// TIA Portal V15.1 export
// export: Created 2024-06-21T08:41:13.9396276Z, ExportSetting WithDefaults, DisplayName Totally Integrated Automation Portal, DisplayVersion V15.1 Update 5, DisplayName TIA Portal Openness, DisplayVersion V15.1 Update 5, DisplayName SINAMICS Startdrive Advanced, DisplayVersion V15.1, DisplayName G130, G150, S120, S150, SINAMICS MV, S210, DisplayVersion V15.1, DisplayName G110M, G120, G120C, G120D, G120P, DisplayVersion V15.1, DisplayName STEP 7 Professional, DisplayVersion V15.1 Update 5, DisplayName STEP 7 Safety, DisplayVersion V15.1, DisplayName WinCC Professional, DisplayVersion V15.1 Update 5, DisplayName SIMATIC Visualization Architect, DisplayVersion V15.1
FUNCTION_BLOCK "LGBBuhlLock"   // FB6630, FBD
TITLE = LGBBuhlLock
{ S7_Optimized_Access := 'TRUE' }
AUTHOR : VCC
FAMILY : Tooling
VERSION : 0.1
// ==================================================
// This module handles a Move Unit with 2 Positions and Contactor
// ==================================================
// stored: AutoNumber false, IsIECCheckEnabled false, IsRetainMemResEnabled false, MemoryReserve 100, SetENOAutomatically False, UDAEnableTagReadback false
   VAR_INPUT
      I_PosSetDet1 { ExternalAccessible := 'False'; ExternalVisible := 'False'; ExternalWritable := 'False'} : Bool;   // Position Set Detection1 (Unlocked)
      I_PosSetDet2 { ExternalAccessible := 'False'; ExternalVisible := 'False'; ExternalWritable := 'False'} : Bool;   // Position Set Detection2 (Unlocked)
      I_PosResDet1 { ExternalAccessible := 'False'; ExternalVisible := 'False'; ExternalWritable := 'False'} : Bool;   // Position Reset Detection1 (Locked)
      I_PosResDet2 { ExternalAccessible := 'False'; ExternalVisible := 'False'; ExternalWritable := 'False'} : Bool;   // Position Reset Detection2 (Locked)
      I_Ready { ExternalAccessible := 'False'; ExternalVisible := 'False'; ExternalWritable := 'False'} : Bool;   // Device Ready
      I_SetBegin { ExternalAccessible := 'False'; ExternalVisible := 'False'; ExternalWritable := 'False'} : Bool;   // Function Set begin selection
      I_ResBegin { ExternalAccessible := 'False'; ExternalVisible := 'False'; ExternalWritable := 'False'} : Bool;   // Function Reset begin selection
      I_PBSet { ExternalAccessible := 'False'; ExternalVisible := 'False'; ExternalWritable := 'False'} : Bool;   // Push button for Set direction (used in manual with button OP panels )
      I_PBReset { ExternalAccessible := 'False'; ExternalVisible := 'False'; ExternalWritable := 'False'} : Bool;   // Push button for Reset direction (used in manual with Pushbutton OP panels)
      I_SetIntlkOK { ExternalAccessible := 'False'; ExternalVisible := 'False'; ExternalWritable := 'False'} : Bool;   // Set Interlock
      I_ResIntlkOK { ExternalAccessible := 'False'; ExternalVisible := 'False'; ExternalWritable := 'False'} : Bool;   // Reset Interlock
      I_SafetyOk { ExternalAccessible := 'False'; ExternalVisible := 'False'; ExternalWritable := 'False'} : Bool;   // Safety Ok
      I_MotorProtection { ExternalAccessible := 'False'; ExternalVisible := 'False'; ExternalWritable := 'False'} : Bool;   // Motor protection
      I_SafetySwitch { ExternalAccessible := 'False'; ExternalVisible := 'False'; ExternalWritable := 'False'} : Bool;   // Safety Switch
      I_ModeScreenChanged { ExternalAccessible := 'False'; ExternalVisible := 'False'; ExternalWritable := 'False'} : Bool;   // Screen Changed
   END_VAR
   VAR_OUTPUT
      O_CmdSet { ExternalAccessible := 'False'; ExternalVisible := 'False'; ExternalWritable := 'False'} : Bool;   // Command to Activate Set movement
      O_CmdRes { ExternalAccessible := 'False'; ExternalVisible := 'False'; ExternalWritable := 'False'} : Bool;   // Command to Activate Reset movement
      O_SumPosSet { ExternalAccessible := 'False'; ExternalVisible := 'False'; ExternalWritable := 'False'} : Bool;   // Summary In Position Set
      O_SumPosRes { ExternalAccessible := 'False'; ExternalVisible := 'False'; ExternalWritable := 'False'} : Bool;   // Summary In Position Reset
      O_FuncRunning { ExternalAccessible := 'False'; ExternalVisible := 'False'; ExternalWritable := 'False'} : Bool;   // Signal that the function is busy
      O_SetFinished { ExternalAccessible := 'False'; ExternalVisible := 'False'; ExternalWritable := 'False'} : Bool;   // Function Set finished
      O_ResFinished { ExternalAccessible := 'False'; ExternalVisible := 'False'; ExternalWritable := 'False'} : Bool;   // Function Reset finished
      O_AlarmABCondition { ExternalAccessible := 'False'; ExternalVisible := 'False'; ExternalWritable := 'False'} : Bool;   // Alarm AB Condition
      O_AlarmA { ExternalAccessible := 'False'; ExternalVisible := 'False'; ExternalWritable := 'False'} : Bool;   // Alarm A
      O_AlarmB { ExternalAccessible := 'False'; ExternalVisible := 'False'; ExternalWritable := 'False'} : Bool;   // Alarm B
      O_AlarmC { ExternalAccessible := 'False'; ExternalVisible := 'False'; ExternalWritable := 'False'} : Bool;   // Alarm C
      O_AlarmD { ExternalAccessible := 'False'; ExternalVisible := 'False'; ExternalWritable := 'False'} : Bool;   // Alarm D
      H_AlarmDWord { ExternalAccessible := 'False'; ExternalVisible := 'False'; ExternalWritable := 'False'} : DWord;   // HMI Alarm Word
   END_VAR
   VAR_IN_OUT
      IO_ModeSelector : Struct   // Mode Selector
         AutoSel : Bool;
         AllAutoSel : Bool;
         StepSel : Bool;
         HomeRunSel : Bool;
         ManualSel : Bool;
         ForcedManActSel : Bool;
         PBSetSel : Bool;
         PBResetSel : Bool;
         StartPBSel : Bool;
         AlarmResetPBSel : Bool;
         ResetTMSel : Bool;
         ResetSeqSel : Bool;
         CycleFinishedSel : Bool;
         HomeRunRedoSel : Bool;
         HomeRunWorkDoneSel : Bool;
         ResetSafetyInputSel : Bool;
      END_STRUCT;
      IO_Alarm : "Alarm";   // Alarm
      C_MovConfig : "MovConfig";   // Config
      H_HMI : "H_HMI";   // Animation
      H_GBBuhlLock : "H_GBBuhlLock";   // Animation
   END_VAR
   VAR
      Modes { ExternalAccessible := 'False'; ExternalVisible := 'False'; ExternalWritable := 'False'} : "Modes";   // Modes
      H_FncSelInHMI { ExternalAccessible := 'False'; ExternalVisible := 'False'; ExternalWritable := 'False'} : Bool;
      AA_MotorProtection { ExternalAccessible := 'False'; ExternalVisible := 'False'; ExternalWritable := 'False'} : Bool;   // Motorprotection Not Ok / Motorprotection Tripped
      AA_SafetySwitch { ExternalAccessible := 'False'; ExternalVisible := 'False'; ExternalWritable := 'False'} : Bool;   // Safety Switch Not Ok
      AB_KeepPosSetAlm { ExternalAccessible := 'False'; ExternalVisible := 'False'; ExternalWritable := 'False'} : Bool;   // Lost Set Position / Alarm Keep Position Set
      AB_KeepPosResAlm { ExternalAccessible := 'False'; ExternalVisible := 'False'; ExternalWritable := 'False'} : Bool;   // Lost Reset Position / Alarm Keep Position Reset
      AB_OvtSetAlm { ExternalAccessible := 'False'; ExternalVisible := 'False'; ExternalWritable := 'False'} : Bool;   // TimeOut Set Direction / Timeout Set
      AB_OvtResAlm { ExternalAccessible := 'False'; ExternalVisible := 'False'; ExternalWritable := 'False'} : Bool;   // TimeOut Reset Direction / Timeout Reset
      AB_TwoDetAlm { ExternalAccessible := 'False'; ExternalVisible := 'False'; ExternalWritable := 'False'} : Bool;   // Detection Set & Reset Activated Simultaneously / Set Reset Activated Simultaneously
      AC_KeepPosSetAlm { ExternalAccessible := 'False'; ExternalVisible := 'False'; ExternalWritable := 'False'} : Bool;   // Lost Set Position / Alarm Keep Position Set
      AC_KeepPosResAlm { ExternalAccessible := 'False'; ExternalVisible := 'False'; ExternalWritable := 'False'} : Bool;   // Lost Reset Position / Alarm Keep Position Reset
      AC_OvtSetAlm { ExternalAccessible := 'False'; ExternalVisible := 'False'; ExternalWritable := 'False'} : Bool;   // TimeOut Set Direction / Timeout Set
      AC_OvtResAlm { ExternalAccessible := 'False'; ExternalVisible := 'False'; ExternalWritable := 'False'} : Bool;   // TimeOut Reset Direction / Timeout Reset
      AC_TwoDetAlm { ExternalAccessible := 'False'; ExternalVisible := 'False'; ExternalWritable := 'False'} : Bool;   // Detection Set & Reset Activated Simultaneously / Set Reset Activated Simultaneously
      AD_OvtSetWarn { ExternalAccessible := 'False'; ExternalVisible := 'False'; ExternalWritable := 'False'} : Bool;   // TimeOut Set Direction / Timeout Set
      AD_OvtResWarn { ExternalAccessible := 'False'; ExternalVisible := 'False'; ExternalWritable := 'False'} : Bool;   // TimeOut Reset Direction / Timeout Reset
      AD_IntlkSetAlm { ExternalAccessible := 'False'; ExternalVisible := 'False'; ExternalWritable := 'False'} : Bool;   // Interlock Set
      AD_IntlkResAlm { ExternalAccessible := 'False'; ExternalVisible := 'False'; ExternalWritable := 'False'} : Bool;   // Interlock Reset
      AC_NotReadyAlm { ExternalAccessible := 'False'; ExternalVisible := 'False'; ExternalWritable := 'False'} : Bool;   // Not Ready To Run
      AC_ConfigCalibrationAlm { ExternalAccessible := 'False'; ExternalVisible := 'False'; ExternalWritable := 'False'} : Bool;   // The Config values for Warming/Alarm time must be ALL zero or ALL different from zero
      AD_CalibrationWarn { ExternalAccessible := 'False'; ExternalVisible := 'False'; ExternalWritable := 'False'} : Bool;   // No High speed selected so Calibration is not possible
      CmdSet { ExternalAccessible := 'False'; ExternalVisible := 'False'; ExternalWritable := 'False'} : Bool;   // Command set
      CmdRes { ExternalAccessible := 'False'; ExternalVisible := 'False'; ExternalWritable := 'False'} : Bool;   // DCommand Reset
      SetPos { ExternalAccessible := 'False'; ExternalVisible := 'False'; ExternalWritable := 'False'} : Bool;   // Set Position
      ResPos { ExternalAccessible := 'False'; ExternalVisible := 'False'; ExternalWritable := 'False'} : Bool;   // Reset Position
      AlarmA { ExternalAccessible := 'False'; ExternalVisible := 'False'; ExternalWritable := 'False'} : Bool;   // Summation Alarm A
      AlarmB { ExternalAccessible := 'False'; ExternalVisible := 'False'; ExternalWritable := 'False'} : Bool;   // Summation Alarm B
      AlarmC { ExternalAccessible := 'False'; ExternalVisible := 'False'; ExternalWritable := 'False'} : Bool;   // Summation Alarm C
      AlarmD { ExternalAccessible := 'False'; ExternalVisible := 'False'; ExternalWritable := 'False'} : Bool;   // Summation Alarm D
      FuncRunning { ExternalAccessible := 'False'; ExternalVisible := 'False'; ExternalWritable := 'False'} : Bool;   // Function running
      MovFuncAlmCond { ExternalAccessible := 'False'; ExternalVisible := 'False'; ExternalWritable := 'False'} : Bool;   // Move function Alarm Condition
      StopPosAlmCond { ExternalAccessible := 'False'; ExternalVisible := 'False'; ExternalWritable := 'False'} : Bool;   // Stop posistion Alarm Condition
      KeepPosSetAlm { ExternalAccessible := 'False'; ExternalVisible := 'False'; ExternalWritable := 'False'} : Bool;   // Keep Position Set Alarm
      KeepPosResAlm { ExternalAccessible := 'False'; ExternalVisible := 'False'; ExternalWritable := 'False'} : Bool;   // Keep Position Reset Alarm
      OvtSetAlm { ExternalAccessible := 'False'; ExternalVisible := 'False'; ExternalWritable := 'False'} : Bool;   // Overtime set Alarm
      OvtResAlm { ExternalAccessible := 'False'; ExternalVisible := 'False'; ExternalWritable := 'False'} : Bool;   // Overtime Reset Alarm
      TwoDetAlm { ExternalAccessible := 'False'; ExternalVisible := 'False'; ExternalWritable := 'False'} : Bool;   // Two detection Alarm
      OutOfUse { ExternalAccessible := 'False'; ExternalVisible := 'False'; ExternalWritable := 'False'} : Bool;   // Out of use
      AlarmABCondition { ExternalAccessible := 'False'; ExternalVisible := 'False'; ExternalWritable := 'False'} : Bool;   // Alarm AB Condition
      ContactorSet { ExternalAccessible := 'False'; ExternalVisible := 'False'; ExternalWritable := 'False'} : Bool;   // Contactor Set
      ContactorRes { ExternalAccessible := 'False'; ExternalVisible := 'False'; ExternalWritable := 'False'} : Bool;   // Contactor Reset
      MotorLoopAlmCond { ExternalAccessible := 'False'; ExternalVisible := 'False'; ExternalWritable := 'False'} : Bool;   // Motor loop Alarm condition
      MotorLoopActive { ExternalAccessible := 'False'; ExternalVisible := 'False'; ExternalWritable := 'False'} : Bool;   // Motor Loop Active
      ManReqSet { ExternalAccessible := 'False'; ExternalVisible := 'False'; ExternalWritable := 'False'} : Bool;   // In Manual AND Request Maintenance door
      ManReqReset { ExternalAccessible := 'False'; ExternalVisible := 'False'; ExternalWritable := 'False'} : Bool;   // In Manual AND No Request Maintenance door
      MovFunc2Pos { ExternalAccessible := 'False'; ExternalVisible := 'False'; ExternalWritable := 'False'} : "LMovFnc2Pos";   // FB
      StopPos { ExternalAccessible := 'False'; ExternalVisible := 'False'; ExternalWritable := 'False'} : "L2StopPos";   // FB
      _Motor { ExternalAccessible := 'False'; ExternalVisible := 'False'; ExternalWritable := 'False'} : "LGBMotor2W1S-C";   // FB
      PosSetDelayTimer { ExternalAccessible := 'False'; ExternalVisible := 'False'; ExternalWritable := 'False'} : "LTimer";   // FB
      PosResDelayTimer { ExternalAccessible := 'False'; ExternalVisible := 'False'; ExternalWritable := 'False'} : "LTimer";   // FB
      TP_ManReqSet { ExternalAccessible := 'False'; ExternalVisible := 'False'; ExternalWritable := 'False'} : TP_TIME;   // Timer
      TP_ManReqReset { ExternalAccessible := 'False'; ExternalVisible := 'False'; ExternalWritable := 'False'} : TP_TIME;   // Timer
   END_VAR
   VAR_TEMP
      H_HMITemp : "H_HMI";   // Temp
   END_VAR
   VAR_TEMP   // added for the SCL form of the ladder/FBD networks
      _w1 : Bool;
   END_VAR
BEGIN

REGION Network 1: **** 1 - Inputs **** HMI Commands
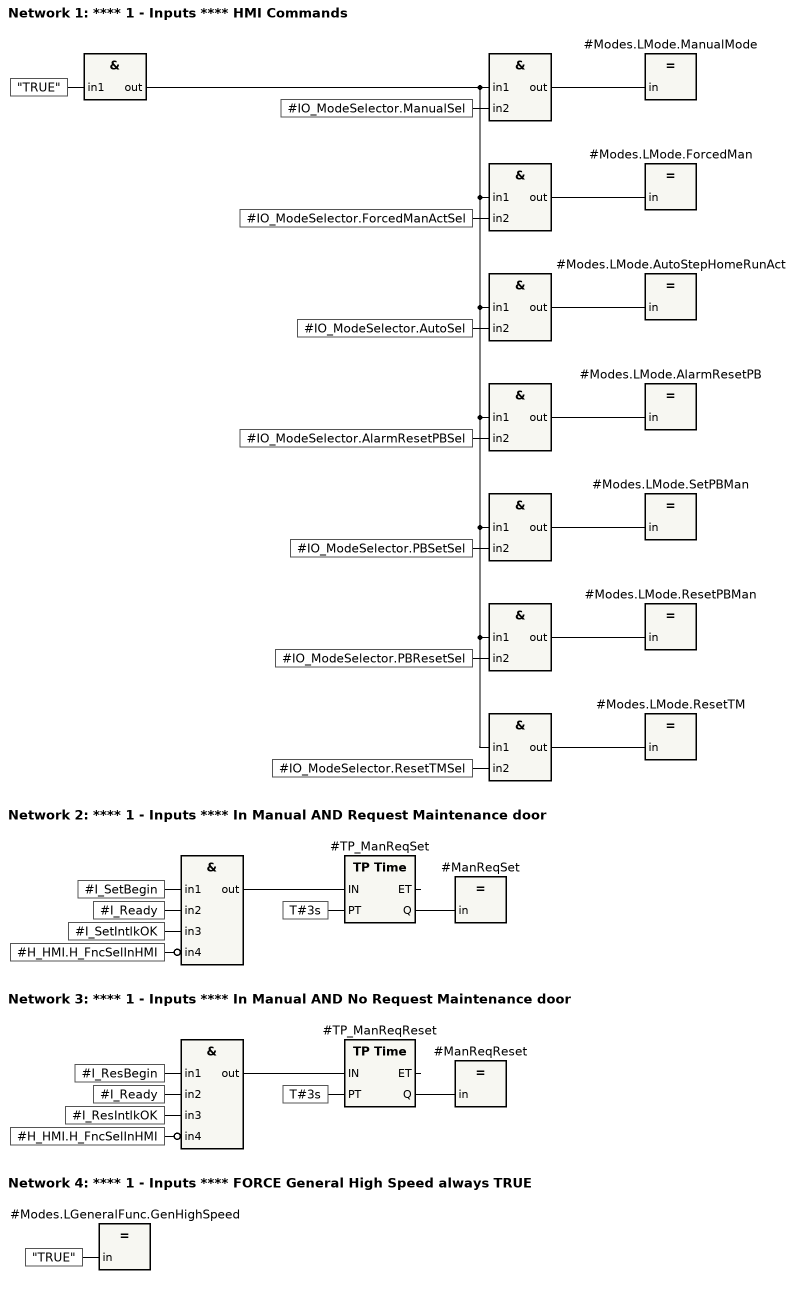
   #Modes.LMode.ManualMode := "TRUE" AND #IO_ModeSelector.ManualSel;
   #Modes.LMode.ForcedMan := "TRUE" AND #IO_ModeSelector.ForcedManActSel;
   #Modes.LMode.AutoStepHomeRunAct := "TRUE" AND #IO_ModeSelector.AutoSel;
   #Modes.LMode.AlarmResetPB := "TRUE" AND #IO_ModeSelector.AlarmResetPBSel;
   #Modes.LMode.SetPBMan := "TRUE" AND #IO_ModeSelector.PBSetSel;
   #Modes.LMode.ResetPBMan := "TRUE" AND #IO_ModeSelector.PBResetSel;
   #Modes.LMode.ResetTM := "TRUE" AND #IO_ModeSelector.ResetTMSel;
END_REGION

REGION Network 2: **** 1 - Inputs **** In Manual AND Request Maintenance door
   #TP_ManReqSet(IN := #I_SetBegin AND #I_Ready AND #I_SetIntlkOK AND NOT #H_HMI.H_FncSelInHMI, PT := T#3s);   // TP
   #ManReqSet := #TP_ManReqSet.Q;
END_REGION

REGION Network 3: **** 1 - Inputs **** In Manual AND No Request Maintenance door
   #TP_ManReqReset(IN := #I_ResBegin AND #I_Ready AND #I_ResIntlkOK AND NOT #H_HMI.H_FncSelInHMI, PT := T#3s);   // TP
   #ManReqReset := #TP_ManReqReset.Q;
END_REGION

REGION Network 4: **** 1 - Inputs **** FORCE General High Speed always TRUE
   #Modes.LGeneralFunc.GenHighSpeed := "TRUE";
END_REGION

REGION Network 5: **** 2.2 - Alarms - Alarm Generation **** Two Detection B Alarm
   // Two Detection B Alarm
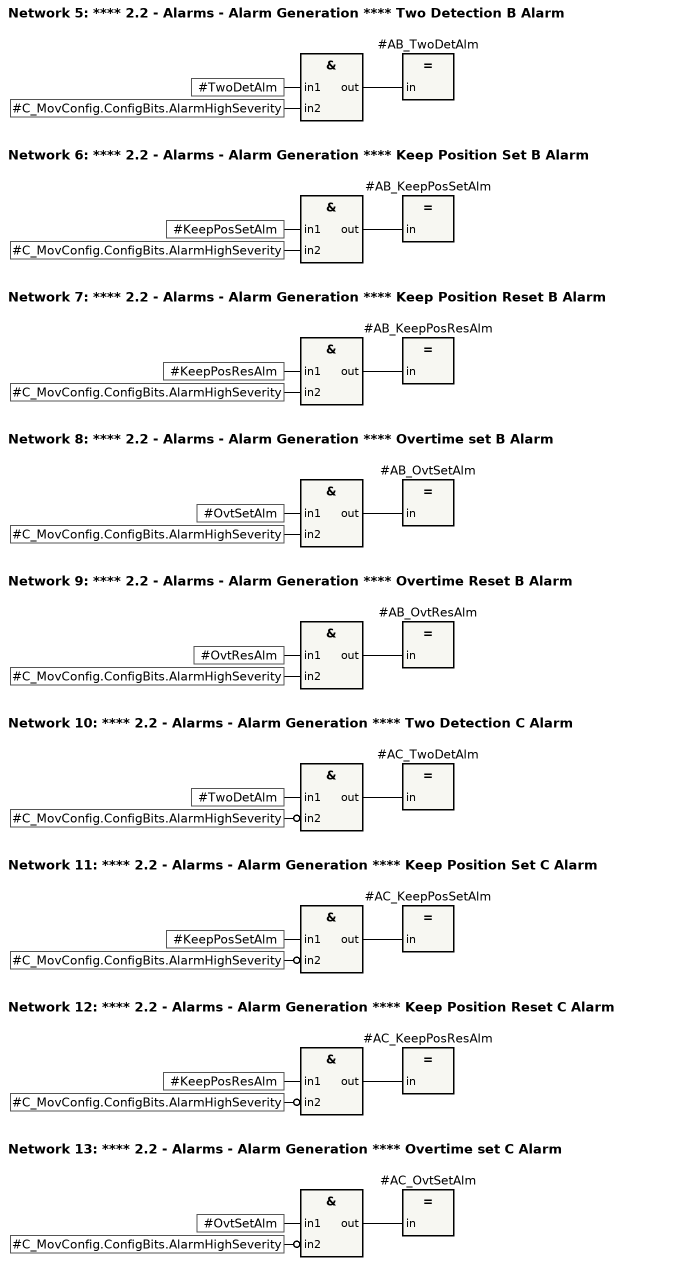
   #AB_TwoDetAlm := #TwoDetAlm AND #C_MovConfig.ConfigBits.AlarmHighSeverity;
END_REGION

REGION Network 6: **** 2.2 - Alarms - Alarm Generation **** Keep Position Set B Alarm
   // Keep Position Set B Alarm
   #AB_KeepPosSetAlm := #KeepPosSetAlm AND #C_MovConfig.ConfigBits.AlarmHighSeverity;
END_REGION

REGION Network 7: **** 2.2 - Alarms - Alarm Generation **** Keep Position Reset B Alarm
   // Keep Position Reset B Alarm
   #AB_KeepPosResAlm := #KeepPosResAlm AND #C_MovConfig.ConfigBits.AlarmHighSeverity;
END_REGION

REGION Network 8: **** 2.2 - Alarms - Alarm Generation **** Overtime set B Alarm
   // Overtime set B Alarm
   #AB_OvtSetAlm := #OvtSetAlm AND #C_MovConfig.ConfigBits.AlarmHighSeverity;
END_REGION

REGION Network 9: **** 2.2 - Alarms - Alarm Generation **** Overtime Reset B Alarm
   // Overtime Reset B Alarm
   #AB_OvtResAlm := #OvtResAlm AND #C_MovConfig.ConfigBits.AlarmHighSeverity;
END_REGION

REGION Network 10: **** 2.2 - Alarms - Alarm Generation **** Two Detection C Alarm
   // Two Detection C Alarm
   #AC_TwoDetAlm := #TwoDetAlm AND NOT #C_MovConfig.ConfigBits.AlarmHighSeverity;
END_REGION

REGION Network 11: **** 2.2 - Alarms - Alarm Generation **** Keep Position Set C Alarm
   // Keep Position Set C Alarm
   #AC_KeepPosSetAlm := #KeepPosSetAlm AND NOT #C_MovConfig.ConfigBits.AlarmHighSeverity;
END_REGION

REGION Network 12: **** 2.2 - Alarms - Alarm Generation **** Keep Position Reset C Alarm
   // Keep Position Reset C Alarm
   #AC_KeepPosResAlm := #KeepPosResAlm AND NOT #C_MovConfig.ConfigBits.AlarmHighSeverity;
END_REGION

REGION Network 13: **** 2.2 - Alarms - Alarm Generation **** Overtime set C Alarm
   // Overtime set C Alarm
   #AC_OvtSetAlm := #OvtSetAlm AND NOT #C_MovConfig.ConfigBits.AlarmHighSeverity;
END_REGION

REGION Network 14: **** 2.2 - Alarms - Alarm Generation **** Overtime Reset C Alarm
   // Overtime Reset C Alarm
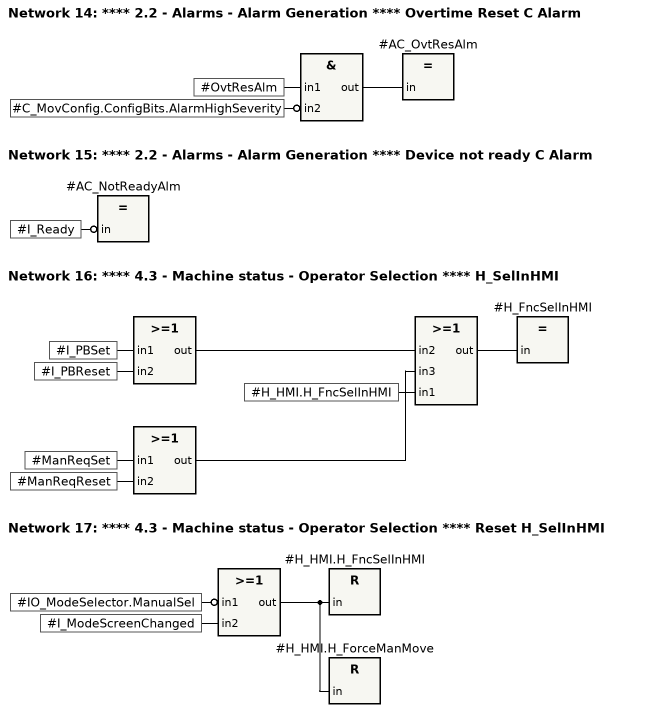
   #AC_OvtResAlm := #OvtResAlm AND NOT #C_MovConfig.ConfigBits.AlarmHighSeverity;
END_REGION

REGION Network 15: **** 2.2 - Alarms - Alarm Generation **** Device not ready C Alarm
   // Device not ready C Alarm
   #AC_NotReadyAlm := NOT #I_Ready;
END_REGION

REGION Network 16: **** 4.3 - Machine status - Operator Selection **** H_SelInHMI
   #H_FncSelInHMI := #I_PBSet OR #I_PBReset OR #ManReqSet OR #ManReqReset OR #H_HMI.H_FncSelInHMI;
END_REGION

REGION Network 17: **** 4.3 - Machine status - Operator Selection **** Reset H_SelInHMI
   // Reset H_SelInHMI
   IF NOT #IO_ModeSelector.ManualSel OR #I_ModeScreenChanged THEN
       #H_HMI.H_FncSelInHMI := FALSE;
       #H_HMI.H_ForceManMove := FALSE;
   END_IF;
END_REGION

REGION Network 18: **** 4.6 - Machine Status - Indication **** Icon Animation
   // Icon Animation
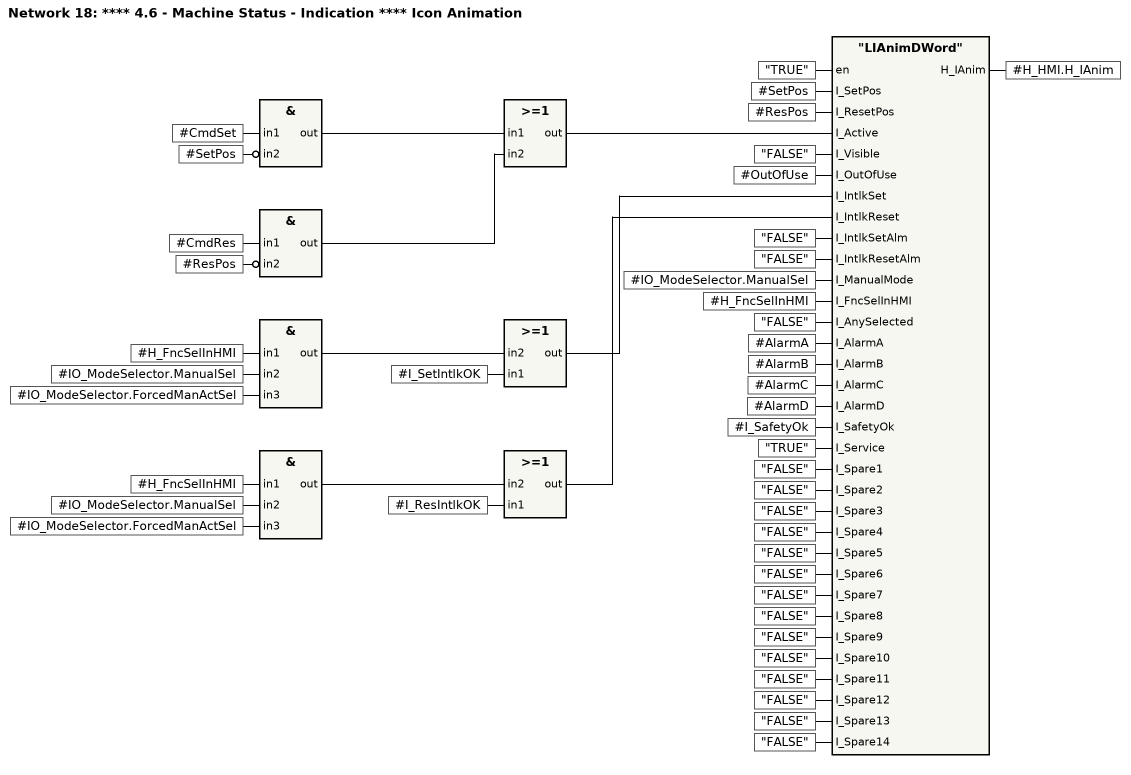
   IF "TRUE" THEN
       "LIAnimDWord"(I_SetPos := #SetPos,
                     I_ResetPos := #ResPos,
                     I_Active := (#CmdSet AND NOT #SetPos) OR (#CmdRes AND NOT #ResPos),
                     I_Visible := "FALSE",
                     I_OutOfUse := #OutOfUse,
                     I_IntlkSet := (#H_FncSelInHMI AND #IO_ModeSelector.ManualSel AND #IO_ModeSelector.ForcedManActSel) OR #I_SetIntlkOK,
                     I_IntlkReset := (#H_FncSelInHMI AND #IO_ModeSelector.ManualSel AND #IO_ModeSelector.ForcedManActSel) OR #I_ResIntlkOK,
                     I_IntlkSetAlm := "FALSE",
                     I_IntlkResetAlm := "FALSE",
                     I_ManualMode := #IO_ModeSelector.ManualSel,
                     I_FncSelInHMI := #H_FncSelInHMI,
                     I_AnySelected := "FALSE",
                     I_AlarmA := #AlarmA,
                     I_AlarmB := #AlarmB,
                     I_AlarmC := #AlarmC,
                     I_AlarmD := #AlarmD,
                     I_SafetyOk := #I_SafetyOk,
                     I_Service := "TRUE",
                     I_Spare1 := "FALSE",
                     I_Spare2 := "FALSE",
                     I_Spare3 := "FALSE",
                     I_Spare4 := "FALSE",
                     I_Spare5 := "FALSE",
                     I_Spare6 := "FALSE",
                     I_Spare7 := "FALSE",
                     I_Spare8 := "FALSE",
                     I_Spare9 := "FALSE",
                     I_Spare10 := "FALSE",
                     I_Spare11 := "FALSE",
                     I_Spare12 := "FALSE",
                     I_Spare13 := "FALSE",
                     I_Spare14 := "FALSE",
                     H_IAnim => #H_HMI.H_IAnim);
   END_IF;
END_REGION

REGION Network 19: **** 4.6 - Machine Status - Indication **** Icon Animation SetDet1
   // Icon Animation
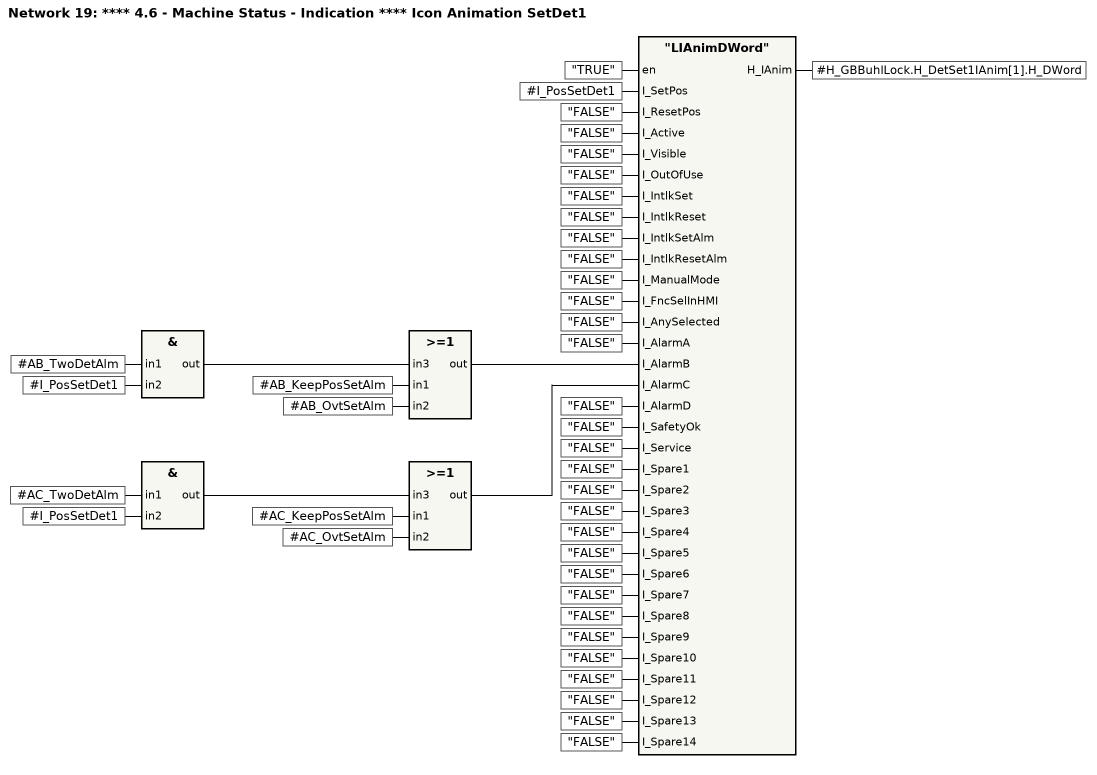
   IF "TRUE" THEN
       "LIAnimDWord"(I_SetPos := #I_PosSetDet1,
                     I_ResetPos := "FALSE",
                     I_Active := "FALSE",
                     I_Visible := "FALSE",
                     I_OutOfUse := "FALSE",
                     I_IntlkSet := "FALSE",
                     I_IntlkReset := "FALSE",
                     I_IntlkSetAlm := "FALSE",
                     I_IntlkResetAlm := "FALSE",
                     I_ManualMode := "FALSE",
                     I_FncSelInHMI := "FALSE",
                     I_AnySelected := "FALSE",
                     I_AlarmA := "FALSE",
                     I_AlarmB := (#AB_TwoDetAlm AND #I_PosSetDet1) OR #AB_KeepPosSetAlm OR #AB_OvtSetAlm,
                     I_AlarmC := (#AC_TwoDetAlm AND #I_PosSetDet1) OR #AC_KeepPosSetAlm OR #AC_OvtSetAlm,
                     I_AlarmD := "FALSE",
                     I_SafetyOk := "FALSE",
                     I_Service := "FALSE",
                     I_Spare1 := "FALSE",
                     I_Spare2 := "FALSE",
                     I_Spare3 := "FALSE",
                     I_Spare4 := "FALSE",
                     I_Spare5 := "FALSE",
                     I_Spare6 := "FALSE",
                     I_Spare7 := "FALSE",
                     I_Spare8 := "FALSE",
                     I_Spare9 := "FALSE",
                     I_Spare10 := "FALSE",
                     I_Spare11 := "FALSE",
                     I_Spare12 := "FALSE",
                     I_Spare13 := "FALSE",
                     I_Spare14 := "FALSE",
                     H_IAnim => #H_GBBuhlLock.H_DetSet1IAnim[1].H_DWord);
   END_IF;
END_REGION

REGION Network 20: **** 4.6 - Machine Status - Indication **** Icon Animation SetDet2
   // Icon Animation
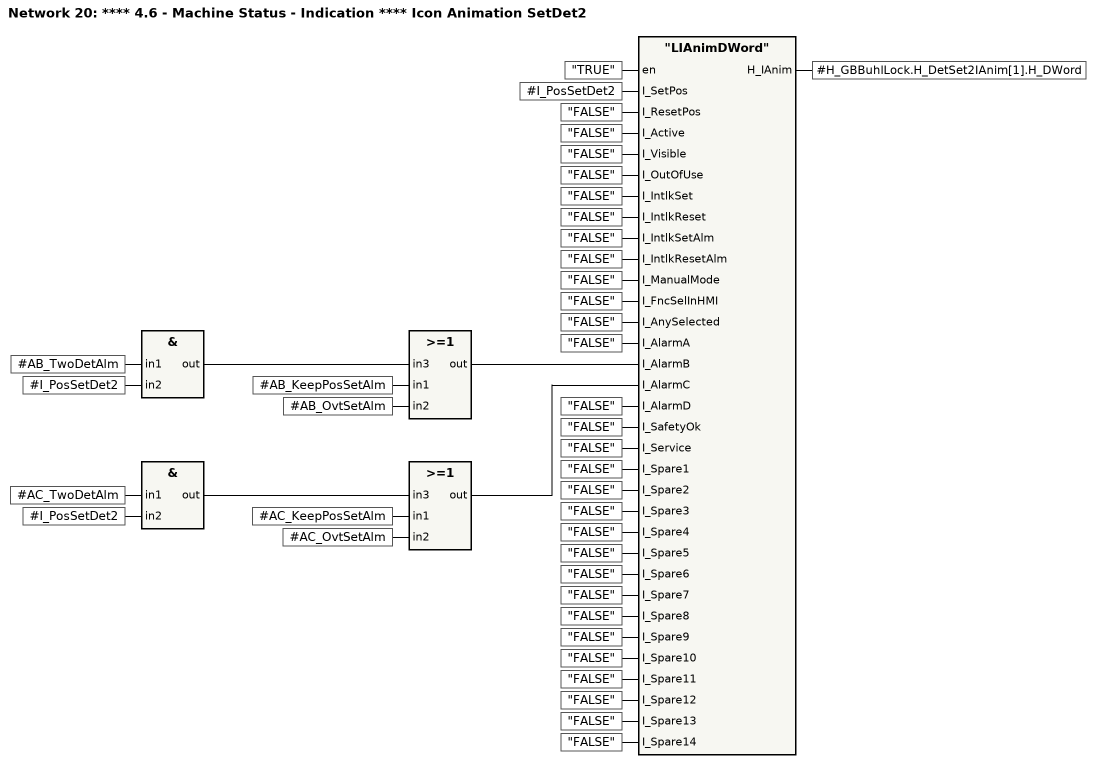
   IF "TRUE" THEN
       "LIAnimDWord"(I_SetPos := #I_PosSetDet2,
                     I_ResetPos := "FALSE",
                     I_Active := "FALSE",
                     I_Visible := "FALSE",
                     I_OutOfUse := "FALSE",
                     I_IntlkSet := "FALSE",
                     I_IntlkReset := "FALSE",
                     I_IntlkSetAlm := "FALSE",
                     I_IntlkResetAlm := "FALSE",
                     I_ManualMode := "FALSE",
                     I_FncSelInHMI := "FALSE",
                     I_AnySelected := "FALSE",
                     I_AlarmA := "FALSE",
                     I_AlarmB := (#AB_TwoDetAlm AND #I_PosSetDet2) OR #AB_KeepPosSetAlm OR #AB_OvtSetAlm,
                     I_AlarmC := (#AC_TwoDetAlm AND #I_PosSetDet2) OR #AC_KeepPosSetAlm OR #AC_OvtSetAlm,
                     I_AlarmD := "FALSE",
                     I_SafetyOk := "FALSE",
                     I_Service := "FALSE",
                     I_Spare1 := "FALSE",
                     I_Spare2 := "FALSE",
                     I_Spare3 := "FALSE",
                     I_Spare4 := "FALSE",
                     I_Spare5 := "FALSE",
                     I_Spare6 := "FALSE",
                     I_Spare7 := "FALSE",
                     I_Spare8 := "FALSE",
                     I_Spare9 := "FALSE",
                     I_Spare10 := "FALSE",
                     I_Spare11 := "FALSE",
                     I_Spare12 := "FALSE",
                     I_Spare13 := "FALSE",
                     I_Spare14 := "FALSE",
                     H_IAnim => #H_GBBuhlLock.H_DetSet2IAnim[1].H_DWord);
   END_IF;
END_REGION

REGION Network 21: **** 4.6 - Machine Status - Indication **** Icon Animation DetRes1
   // Icon Animation
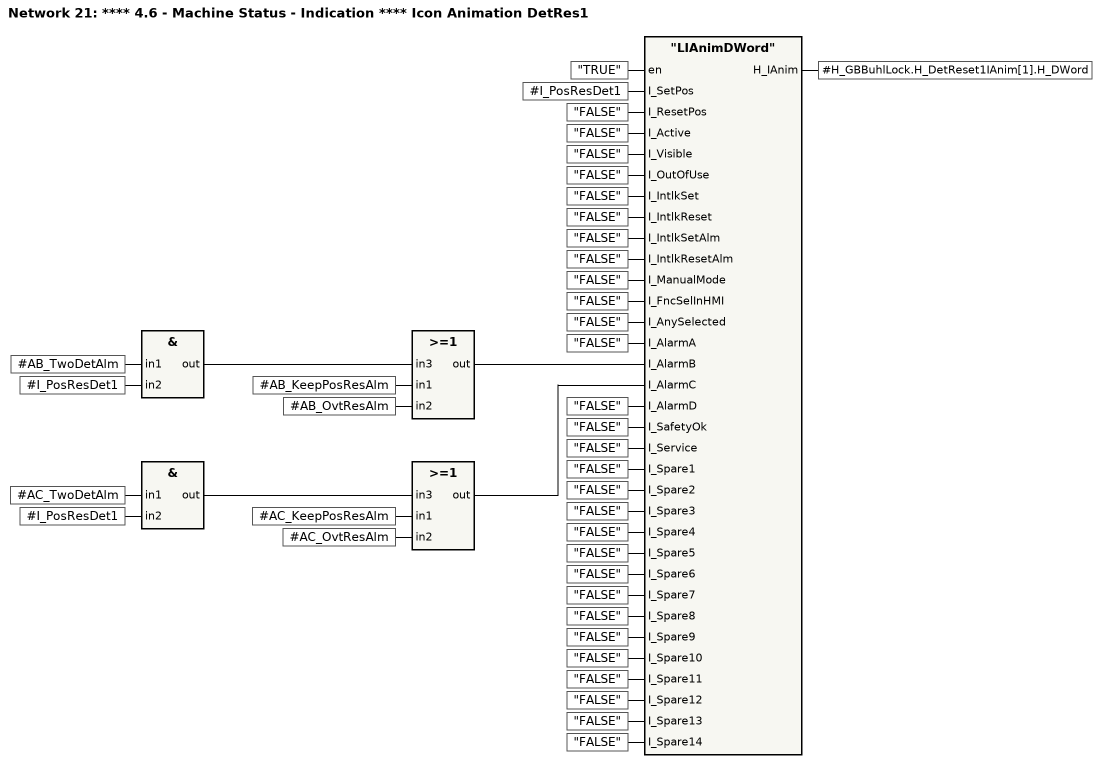
   IF "TRUE" THEN
       "LIAnimDWord"(I_SetPos := #I_PosResDet1,
                     I_ResetPos := "FALSE",
                     I_Active := "FALSE",
                     I_Visible := "FALSE",
                     I_OutOfUse := "FALSE",
                     I_IntlkSet := "FALSE",
                     I_IntlkReset := "FALSE",
                     I_IntlkSetAlm := "FALSE",
                     I_IntlkResetAlm := "FALSE",
                     I_ManualMode := "FALSE",
                     I_FncSelInHMI := "FALSE",
                     I_AnySelected := "FALSE",
                     I_AlarmA := "FALSE",
                     I_AlarmB := (#AB_TwoDetAlm AND #I_PosResDet1) OR #AB_KeepPosResAlm OR #AB_OvtResAlm,
                     I_AlarmC := (#AC_TwoDetAlm AND #I_PosResDet1) OR #AC_KeepPosResAlm OR #AC_OvtResAlm,
                     I_AlarmD := "FALSE",
                     I_SafetyOk := "FALSE",
                     I_Service := "FALSE",
                     I_Spare1 := "FALSE",
                     I_Spare2 := "FALSE",
                     I_Spare3 := "FALSE",
                     I_Spare4 := "FALSE",
                     I_Spare5 := "FALSE",
                     I_Spare6 := "FALSE",
                     I_Spare7 := "FALSE",
                     I_Spare8 := "FALSE",
                     I_Spare9 := "FALSE",
                     I_Spare10 := "FALSE",
                     I_Spare11 := "FALSE",
                     I_Spare12 := "FALSE",
                     I_Spare13 := "FALSE",
                     I_Spare14 := "FALSE",
                     H_IAnim => #H_GBBuhlLock.H_DetReset1IAnim[1].H_DWord);
   END_IF;
END_REGION

REGION Network 22: **** 4.6 - Machine Status - Indication **** Icon Animation DetRes2
   // Icon Animation
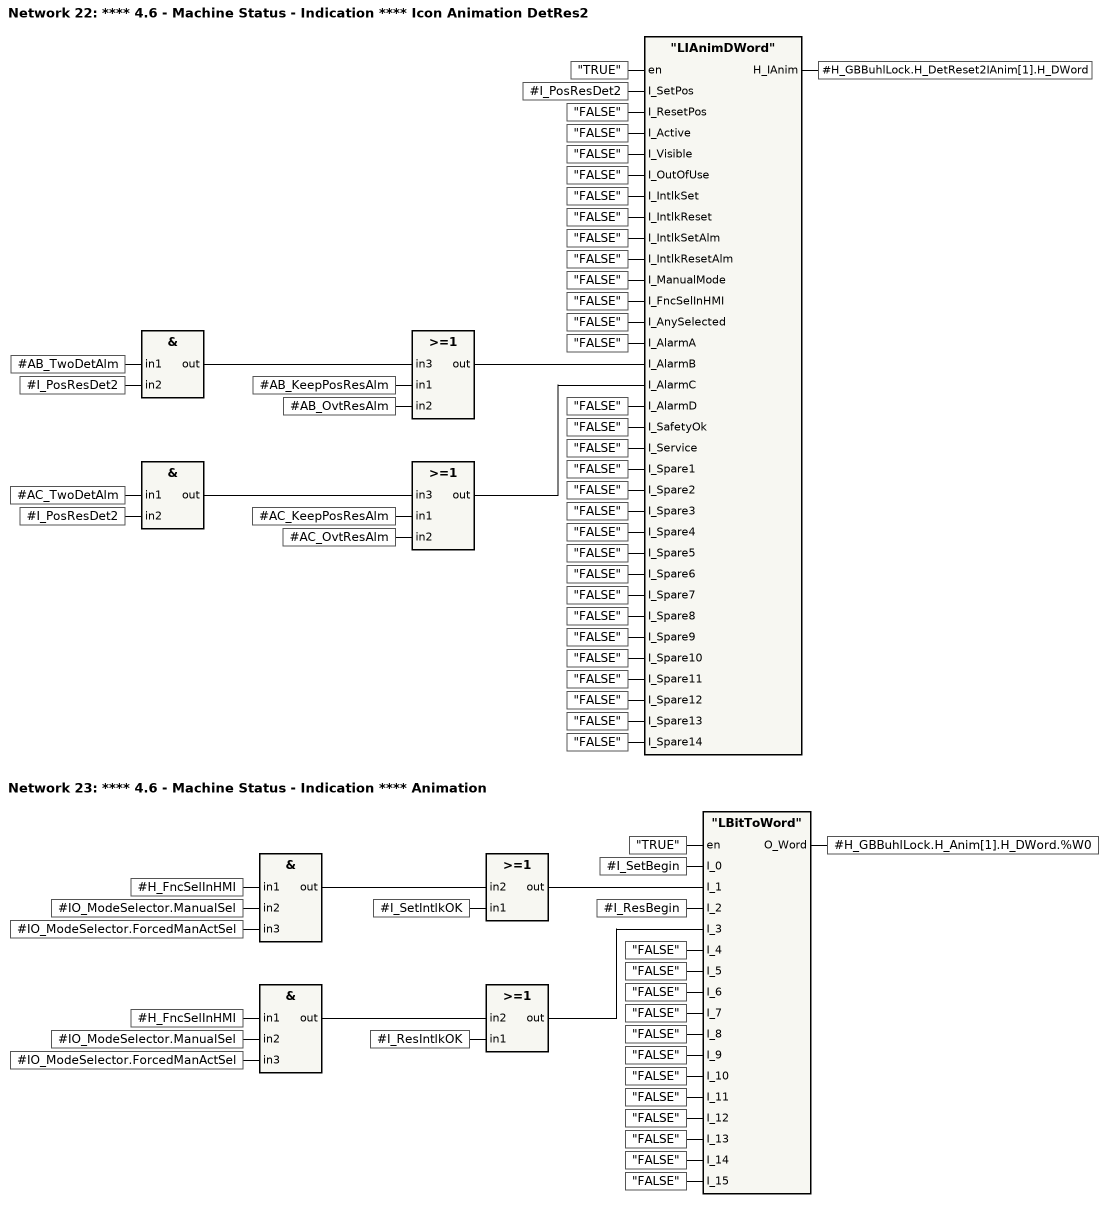
   IF "TRUE" THEN
       "LIAnimDWord"(I_SetPos := #I_PosResDet2,
                     I_ResetPos := "FALSE",
                     I_Active := "FALSE",
                     I_Visible := "FALSE",
                     I_OutOfUse := "FALSE",
                     I_IntlkSet := "FALSE",
                     I_IntlkReset := "FALSE",
                     I_IntlkSetAlm := "FALSE",
                     I_IntlkResetAlm := "FALSE",
                     I_ManualMode := "FALSE",
                     I_FncSelInHMI := "FALSE",
                     I_AnySelected := "FALSE",
                     I_AlarmA := "FALSE",
                     I_AlarmB := (#AB_TwoDetAlm AND #I_PosResDet2) OR #AB_KeepPosResAlm OR #AB_OvtResAlm,
                     I_AlarmC := (#AC_TwoDetAlm AND #I_PosResDet2) OR #AC_KeepPosResAlm OR #AC_OvtResAlm,
                     I_AlarmD := "FALSE",
                     I_SafetyOk := "FALSE",
                     I_Service := "FALSE",
                     I_Spare1 := "FALSE",
                     I_Spare2 := "FALSE",
                     I_Spare3 := "FALSE",
                     I_Spare4 := "FALSE",
                     I_Spare5 := "FALSE",
                     I_Spare6 := "FALSE",
                     I_Spare7 := "FALSE",
                     I_Spare8 := "FALSE",
                     I_Spare9 := "FALSE",
                     I_Spare10 := "FALSE",
                     I_Spare11 := "FALSE",
                     I_Spare12 := "FALSE",
                     I_Spare13 := "FALSE",
                     I_Spare14 := "FALSE",
                     H_IAnim => #H_GBBuhlLock.H_DetReset2IAnim[1].H_DWord);
   END_IF;
END_REGION

REGION Network 23: **** 4.6 - Machine Status - Indication **** Animation
   // Animation
   IF "TRUE" THEN
       "LBitToWord"(I_0 := #I_SetBegin,
                    I_1 := (#H_FncSelInHMI AND #IO_ModeSelector.ManualSel AND #IO_ModeSelector.ForcedManActSel) OR #I_SetIntlkOK,
                    I_2 := #I_ResBegin,
                    I_3 := (#H_FncSelInHMI AND #IO_ModeSelector.ManualSel AND #IO_ModeSelector.ForcedManActSel) OR #I_ResIntlkOK,
                    I_4 := "FALSE",
                    I_5 := "FALSE",
                    I_6 := "FALSE",
                    I_7 := "FALSE",
                    I_8 := "FALSE",
                    I_9 := "FALSE",
                    I_10 := "FALSE",
                    I_11 := "FALSE",
                    I_12 := "FALSE",
                    I_13 := "FALSE",
                    I_14 := "FALSE",
                    I_15 := "FALSE",
                    O_Word => #H_GBBuhlLock.H_Anim[1].H_DWord.%W0);
   END_IF;
END_REGION

REGION Network 24: **** 4.6 - Machine Status - Indication **** Animation
   // Animation
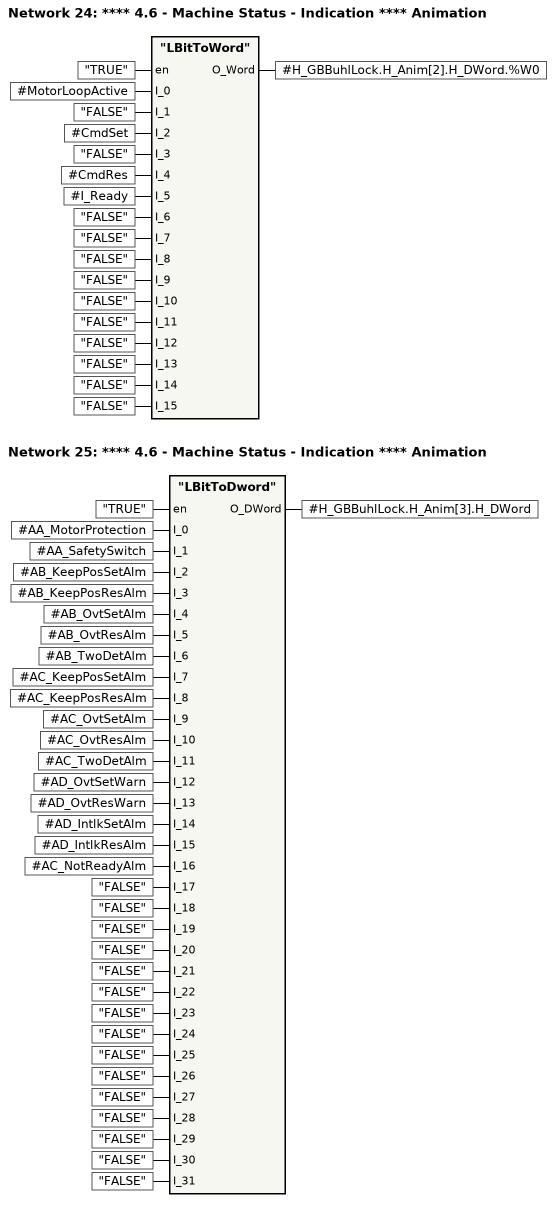
   IF "TRUE" THEN
       "LBitToWord"(I_0 := #MotorLoopActive,
                    I_1 := "FALSE",
                    I_2 := #CmdSet,
                    I_3 := "FALSE",
                    I_4 := #CmdRes,
                    I_5 := #I_Ready,
                    I_6 := "FALSE",
                    I_7 := "FALSE",
                    I_8 := "FALSE",
                    I_9 := "FALSE",
                    I_10 := "FALSE",
                    I_11 := "FALSE",
                    I_12 := "FALSE",
                    I_13 := "FALSE",
                    I_14 := "FALSE",
                    I_15 := "FALSE",
                    O_Word => #H_GBBuhlLock.H_Anim[2].H_DWord.%W0);
   END_IF;
END_REGION

REGION Network 25: **** 4.6 - Machine Status - Indication **** Animation
   // Animation
   IF "TRUE" THEN
       "LBitToDword"(I_0 := #AA_MotorProtection,
                     I_1 := #AA_SafetySwitch,
                     I_2 := #AB_KeepPosSetAlm,
                     I_3 := #AB_KeepPosResAlm,
                     I_4 := #AB_OvtSetAlm,
                     I_5 := #AB_OvtResAlm,
                     I_6 := #AB_TwoDetAlm,
                     I_7 := #AC_KeepPosSetAlm,
                     I_8 := #AC_KeepPosResAlm,
                     I_9 := #AC_OvtSetAlm,
                     I_10 := #AC_OvtResAlm,
                     I_11 := #AC_TwoDetAlm,
                     I_12 := #AD_OvtSetWarn,
                     I_13 := #AD_OvtResWarn,
                     I_14 := #AD_IntlkSetAlm,
                     I_15 := #AD_IntlkResAlm,
                     I_16 := #AC_NotReadyAlm,
                     I_17 := "FALSE",
                     I_18 := "FALSE",
                     I_19 := "FALSE",
                     I_20 := "FALSE",
                     I_21 := "FALSE",
                     I_22 := "FALSE",
                     I_23 := "FALSE",
                     I_24 := "FALSE",
                     I_25 := "FALSE",
                     I_26 := "FALSE",
                     I_27 := "FALSE",
                     I_28 := "FALSE",
                     I_29 := "FALSE",
                     I_30 := "FALSE",
                     I_31 := "FALSE",
                     O_DWord => #H_GBBuhlLock.H_Anim[3].H_DWord);
   END_IF;
END_REGION

REGION Network 26: **** 7.3 - Submodule - Machine **** LMovFunc2Pos
   // LMovFunc2Pos
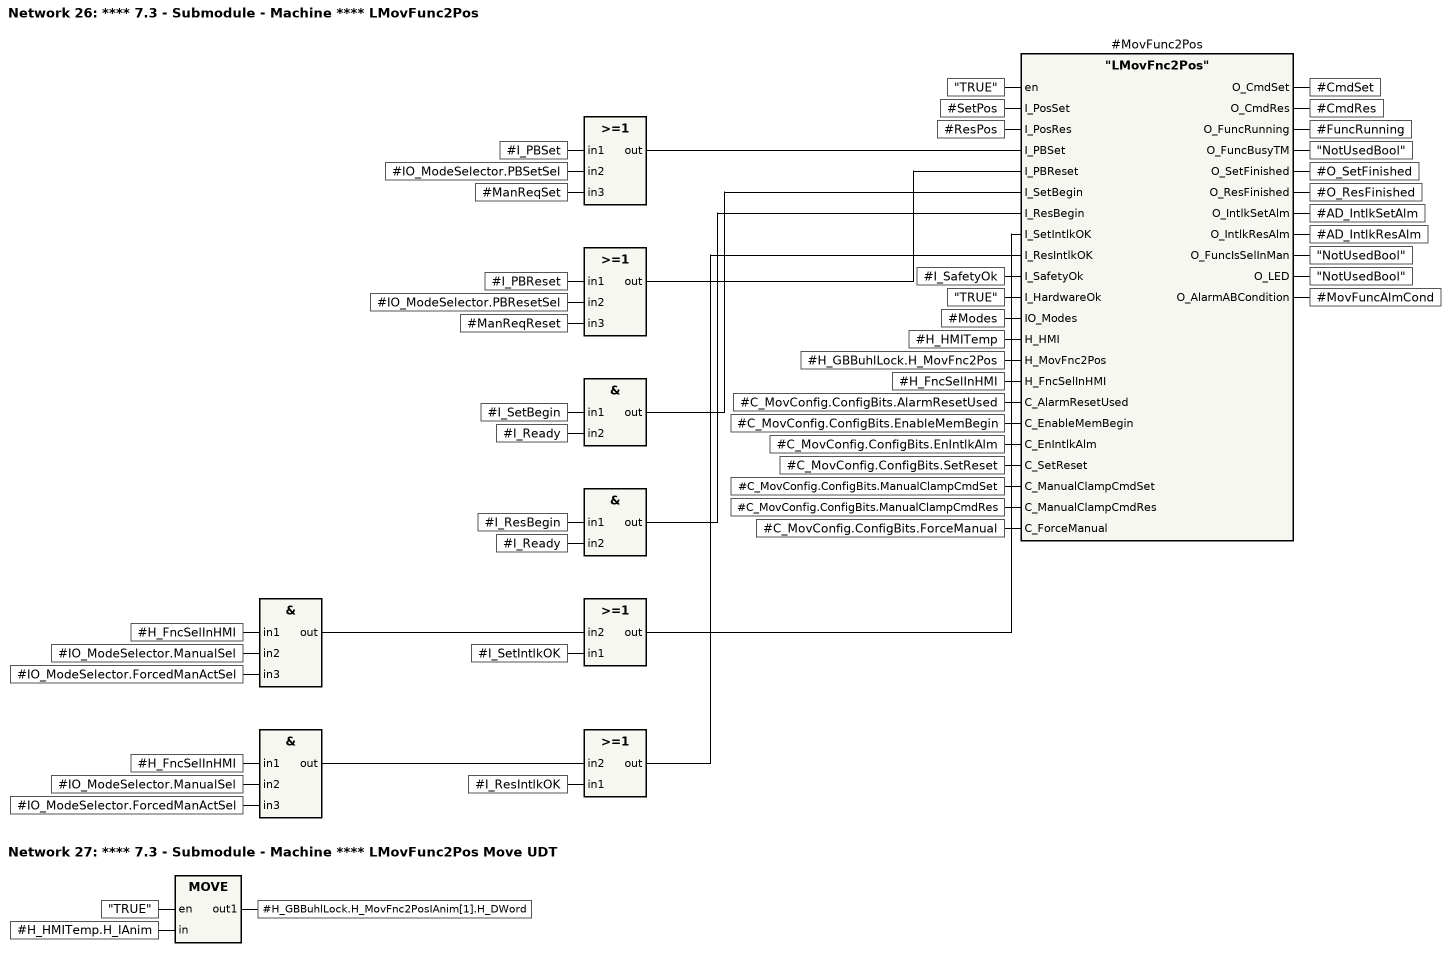
   IF "TRUE" THEN
       #MovFunc2Pos(I_PosSet := #SetPos,   // "LMovFnc2Pos"
                    I_PosRes := #ResPos,
                    I_PBSet := #I_PBSet OR #IO_ModeSelector.PBSetSel OR #ManReqSet,
                    I_PBReset := #I_PBReset OR #IO_ModeSelector.PBResetSel OR #ManReqReset,
                    I_SetBegin := #I_SetBegin AND #I_Ready,
                    I_ResBegin := #I_ResBegin AND #I_Ready,
                    I_SetIntlkOK := (#H_FncSelInHMI AND #IO_ModeSelector.ManualSel AND #IO_ModeSelector.ForcedManActSel) OR #I_SetIntlkOK,
                    I_ResIntlkOK := (#H_FncSelInHMI AND #IO_ModeSelector.ManualSel AND #IO_ModeSelector.ForcedManActSel) OR #I_ResIntlkOK,
                    I_SafetyOk := #I_SafetyOk,
                    I_HardwareOk := "TRUE",
                    IO_Modes := #Modes,
                    H_HMI := #H_HMITemp,
                    H_MovFnc2Pos := #H_GBBuhlLock.H_MovFnc2Pos,
                    H_FncSelInHMI := #H_FncSelInHMI,
                    C_AlarmResetUsed := #C_MovConfig.ConfigBits.AlarmResetUsed,
                    C_EnableMemBegin := #C_MovConfig.ConfigBits.EnableMemBegin,
                    C_EnIntlkAlm := #C_MovConfig.ConfigBits.EnIntlkAlm,
                    C_SetReset := #C_MovConfig.ConfigBits.SetReset,
                    C_ManualClampCmdSet := #C_MovConfig.ConfigBits.ManualClampCmdSet,
                    C_ManualClampCmdRes := #C_MovConfig.ConfigBits.ManualClampCmdRes,
                    C_ForceManual := #C_MovConfig.ConfigBits.ForceManual,
                    O_CmdSet => #CmdSet,
                    O_CmdRes => #CmdRes,
                    O_FuncRunning => #FuncRunning,
                    O_FuncBusyTM => "NotUsedBool",
                    O_SetFinished => #O_SetFinished,
                    O_ResFinished => #O_ResFinished,
                    O_IntlkSetAlm => #AD_IntlkSetAlm,
                    O_IntlkResAlm => #AD_IntlkResAlm,
                    O_FuncIsSelInMan => "NotUsedBool",
                    O_LED => "NotUsedBool",
                    O_AlarmABCondition => #MovFuncAlmCond);
   END_IF;
END_REGION

REGION Network 27: **** 7.3 - Submodule - Machine **** LMovFunc2Pos Move UDT
   // LMovFunc2Pos Move UDT
   IF "TRUE" THEN #H_GBBuhlLock.H_MovFnc2PosIAnim[1].H_DWord := #H_HMITemp.H_IAnim; END_IF;
END_REGION

REGION Network 28: **** 7.3 - Submodule - Machine **** L2StopPos
   // L2StopPos
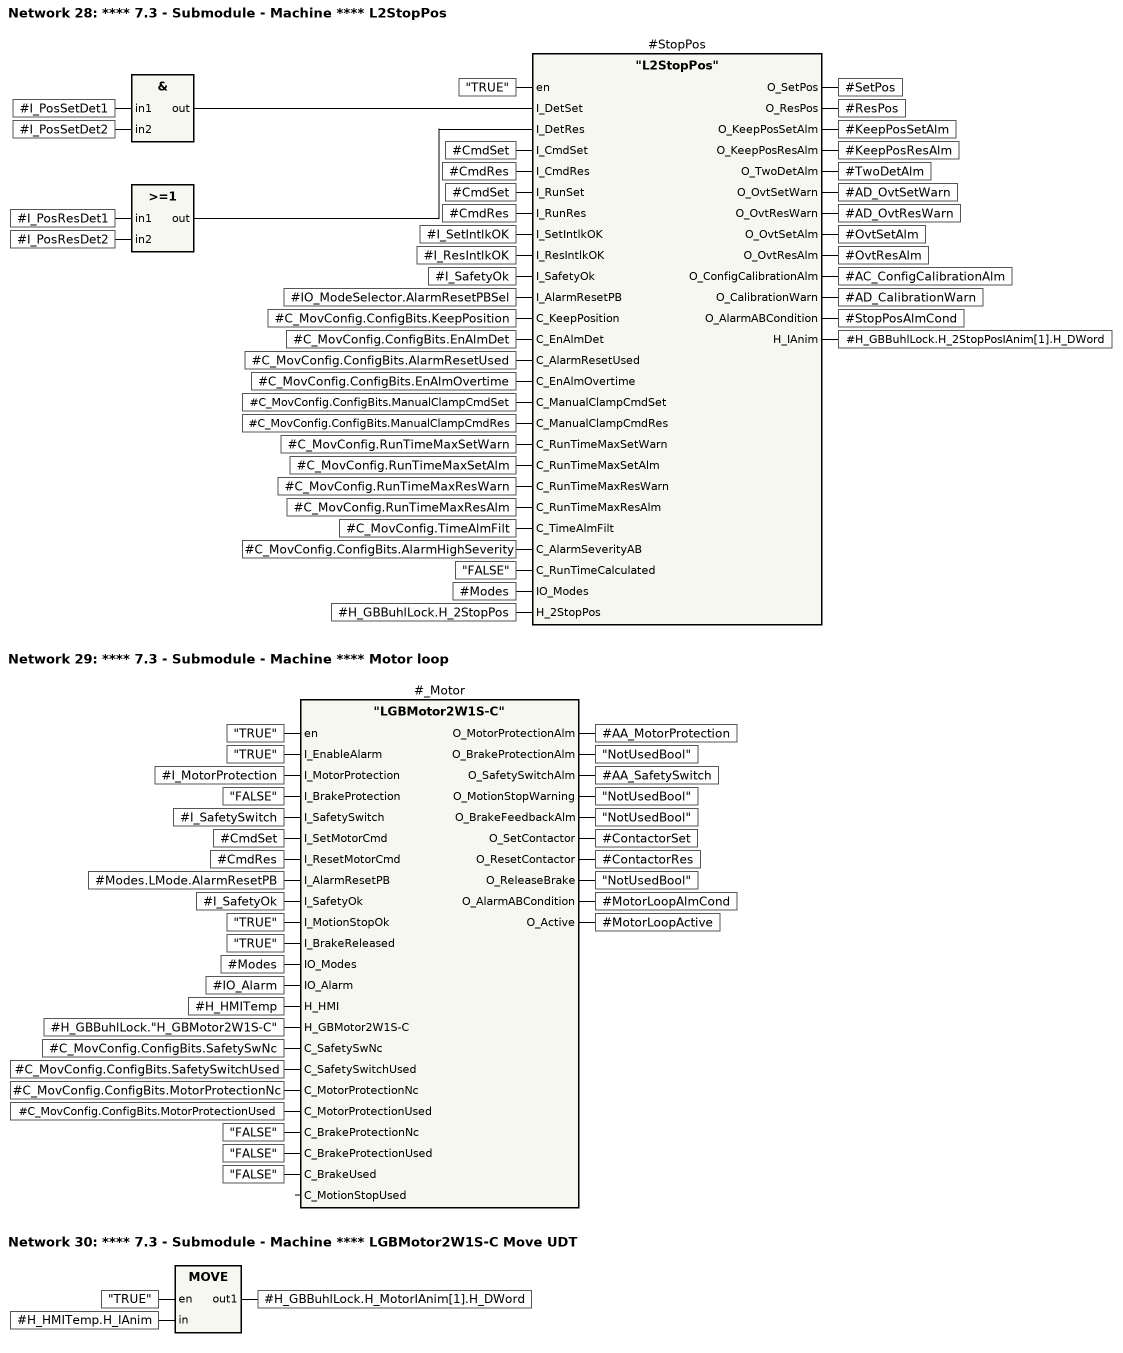
   IF "TRUE" THEN
       #StopPos(I_DetSet := #I_PosSetDet1 AND #I_PosSetDet2,   // "L2StopPos"
                I_DetRes := #I_PosResDet1 OR #I_PosResDet2,
                I_CmdSet := #CmdSet,
                I_CmdRes := #CmdRes,
                I_RunSet := #CmdSet,
                I_RunRes := #CmdRes,
                I_SetIntlkOK := #I_SetIntlkOK,
                I_ResIntlkOK := #I_ResIntlkOK,
                I_SafetyOk := #I_SafetyOk,
                I_AlarmResetPB := #IO_ModeSelector.AlarmResetPBSel,
                C_KeepPosition := #C_MovConfig.ConfigBits.KeepPosition,
                C_EnAlmDet := #C_MovConfig.ConfigBits.EnAlmDet,
                C_AlarmResetUsed := #C_MovConfig.ConfigBits.AlarmResetUsed,
                C_EnAlmOvertime := #C_MovConfig.ConfigBits.EnAlmOvertime,
                C_ManualClampCmdSet := #C_MovConfig.ConfigBits.ManualClampCmdSet,
                C_ManualClampCmdRes := #C_MovConfig.ConfigBits.ManualClampCmdRes,
                C_RunTimeMaxSetWarn := #C_MovConfig.RunTimeMaxSetWarn,
                C_RunTimeMaxSetAlm := #C_MovConfig.RunTimeMaxSetAlm,
                C_RunTimeMaxResWarn := #C_MovConfig.RunTimeMaxResWarn,
                C_RunTimeMaxResAlm := #C_MovConfig.RunTimeMaxResAlm,
                C_TimeAlmFilt := #C_MovConfig.TimeAlmFilt,
                C_AlarmSeverityAB := #C_MovConfig.ConfigBits.AlarmHighSeverity,
                C_RunTimeCalculated := "FALSE",
                IO_Modes := #Modes,
                H_2StopPos := #H_GBBuhlLock.H_2StopPos,
                O_SetPos => #SetPos,
                O_ResPos => #ResPos,
                O_KeepPosSetAlm => #KeepPosSetAlm,
                O_KeepPosResAlm => #KeepPosResAlm,
                O_TwoDetAlm => #TwoDetAlm,
                O_OvtSetWarn => #AD_OvtSetWarn,
                O_OvtResWarn => #AD_OvtResWarn,
                O_OvtSetAlm => #OvtSetAlm,
                O_OvtResAlm => #OvtResAlm,
                O_ConfigCalibrationAlm => #AC_ConfigCalibrationAlm,
                O_CalibrationWarn => #AD_CalibrationWarn,
                O_AlarmABCondition => #StopPosAlmCond,
                H_IAnim => #H_GBBuhlLock.H_2StopPosIAnim[1].H_DWord);
   END_IF;
END_REGION

REGION Network 29: **** 7.3 - Submodule - Machine **** Motor loop
   // Motor loop
   IF "TRUE" THEN
       #_Motor(I_EnableAlarm := "TRUE",   // "LGBMotor2W1S-C"
               I_MotorProtection := #I_MotorProtection,
               I_BrakeProtection := "FALSE",
               I_SafetySwitch := #I_SafetySwitch,
               I_SetMotorCmd := #CmdSet,
               I_ResetMotorCmd := #CmdRes,
               I_AlarmResetPB := #Modes.LMode.AlarmResetPB,
               I_SafetyOk := #I_SafetyOk,
               I_MotionStopOk := "TRUE",
               I_BrakeReleased := "TRUE",
               IO_Modes := #Modes,
               IO_Alarm := #IO_Alarm,
               H_HMI := #H_HMITemp,
               "H_GBMotor2W1S-C" := #H_GBBuhlLock."H_GBMotor2W1S-C",
               C_SafetySwNc := #C_MovConfig.ConfigBits.SafetySwNc,
               C_SafetySwitchUsed := #C_MovConfig.ConfigBits.SafetySwitchUsed,
               C_MotorProtectionNc := #C_MovConfig.ConfigBits.MotorProtectionNc,
               C_MotorProtectionUsed := #C_MovConfig.ConfigBits.MotorProtectionUsed,
               C_BrakeProtectionNc := "FALSE",
               C_BrakeProtectionUsed := "FALSE",
               C_BrakeUsed := "FALSE",
               O_MotorProtectionAlm => #AA_MotorProtection,
               O_BrakeProtectionAlm => "NotUsedBool",
               O_SafetySwitchAlm => #AA_SafetySwitch,
               O_MotionStopWarning => "NotUsedBool",
               O_BrakeFeedbackAlm => "NotUsedBool",
               O_SetContactor => #ContactorSet,
               O_ResetContactor => #ContactorRes,
               O_ReleaseBrake => "NotUsedBool",
               O_AlarmABCondition => #MotorLoopAlmCond,
               O_Active => #MotorLoopActive);
   END_IF;
END_REGION

REGION Network 30: **** 7.3 - Submodule - Machine **** LGBMotor2W1S-C Move UDT
   // LGBMotor2W2S-C Move UDT
   IF "TRUE" THEN #H_GBBuhlLock.H_MotorIAnim[1].H_DWord := #H_HMITemp.H_IAnim; END_IF;
END_REGION

REGION Network 31: **** 8 - Outputs **** Function running
   // Function running
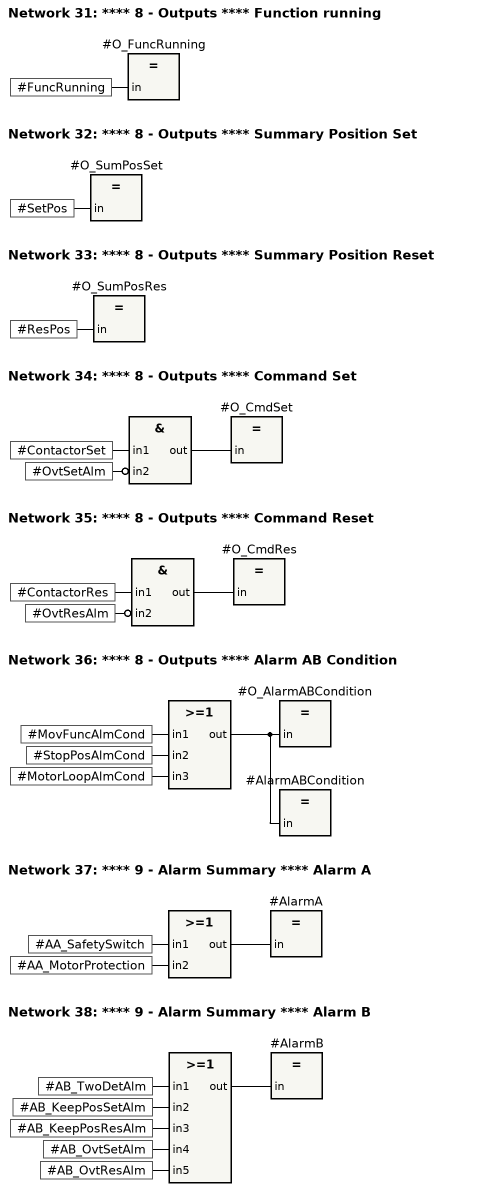
   #O_FuncRunning := #FuncRunning;
END_REGION

REGION Network 32: **** 8 - Outputs **** Summary Position Set
   // Summary Position Set
   #O_SumPosSet := #SetPos;
END_REGION

REGION Network 33: **** 8 - Outputs **** Summary Position Reset
   // Summary Position Reset
   #O_SumPosRes := #ResPos;
END_REGION

REGION Network 34: **** 8 - Outputs **** Command Set
   // Command Set
   #O_CmdSet := #ContactorSet AND NOT #OvtSetAlm;
END_REGION

REGION Network 35: **** 8 - Outputs **** Command Reset
   // Command Reset
   #O_CmdRes := #ContactorRes AND NOT #OvtResAlm;
END_REGION

REGION Network 36: **** 8 - Outputs **** Alarm AB Condition
   // Alarm AB Condition
   #O_AlarmABCondition := #MovFuncAlmCond OR #StopPosAlmCond OR #MotorLoopAlmCond;
   #AlarmABCondition := #O_AlarmABCondition;
END_REGION

REGION Network 37: **** 9 - Alarm Summary **** Alarm A
   // Alarms A
   #AlarmA := #AA_SafetySwitch OR #AA_MotorProtection;
END_REGION

REGION Network 38: **** 9 - Alarm Summary **** Alarm B
   // Alarms B
   #AlarmB := #AB_TwoDetAlm OR #AB_KeepPosSetAlm OR #AB_KeepPosResAlm OR #AB_OvtSetAlm OR #AB_OvtResAlm;
END_REGION

REGION Network 39: **** 9 - Alarm Summary **** Alarm C
   // Alarms C
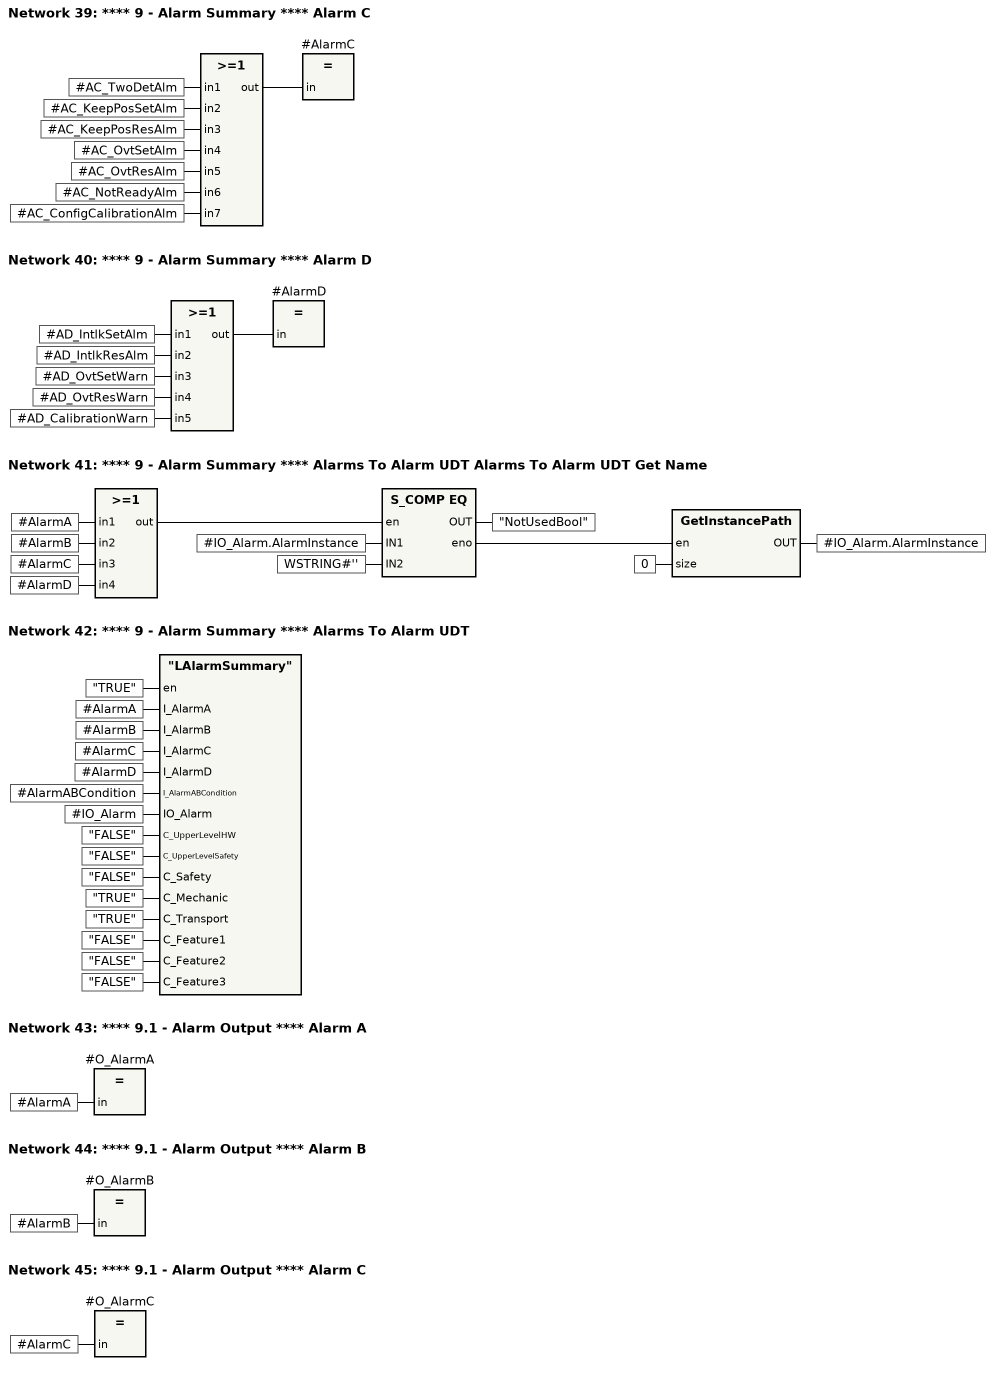
   #AlarmC := #AC_TwoDetAlm OR #AC_KeepPosSetAlm OR #AC_KeepPosResAlm OR #AC_OvtSetAlm OR #AC_OvtResAlm OR #AC_NotReadyAlm OR #AC_ConfigCalibrationAlm;
END_REGION

REGION Network 40: **** 9 - Alarm Summary **** Alarm D
   // Alarms D
   #AlarmD := #AD_IntlkSetAlm OR #AD_IntlkResAlm OR #AD_OvtSetWarn OR #AD_OvtResWarn OR #AD_CalibrationWarn;
END_REGION

REGION Network 41: **** 9 - Alarm Summary **** Alarms To Alarm UDT Alarms To Alarm UDT Get Name
   // Alarm D
   S_COMP(EN := #AlarmA OR #AlarmB OR #AlarmC OR #AlarmD,
          IN1 := #IO_Alarm.AlarmInstance,
          IN2 := WSTRING#'',
          OUT => "NotUsedBool",
          ENO => #_w1);
   IF #_w1 THEN GetInstancePath(size := 0, OUT => #IO_Alarm.AlarmInstance); END_IF;
END_REGION

REGION Network 42: **** 9 - Alarm Summary **** Alarms To Alarm UDT
   // Alarm D
   IF "TRUE" THEN
       "LAlarmSummary"(I_AlarmA := #AlarmA,
                       I_AlarmB := #AlarmB,
                       I_AlarmC := #AlarmC,
                       I_AlarmD := #AlarmD,
                       I_AlarmABCondition := #AlarmABCondition,
                       IO_Alarm := #IO_Alarm,
                       C_UpperLevelHW := "FALSE",
                       C_UpperLevelSafety := "FALSE",
                       C_Safety := "FALSE",
                       C_Mechanic := "TRUE",
                       C_Transport := "TRUE",
                       C_Feature1 := "FALSE",
                       C_Feature2 := "FALSE",
                       C_Feature3 := "FALSE");
   END_IF;
END_REGION

REGION Network 43: **** 9.1 - Alarm Output **** Alarm A
   // Alarms A
   #O_AlarmA := #AlarmA;
END_REGION

REGION Network 44: **** 9.1 - Alarm Output **** Alarm B
   // Alarms B
   #O_AlarmB := #AlarmB;
END_REGION

REGION Network 45: **** 9.1 - Alarm Output **** Alarm C
   // Alarms C
   #O_AlarmC := #AlarmC;
END_REGION

REGION Network 46: **** 9.1 - Alarm Output **** Alarm D
   // Alarms D
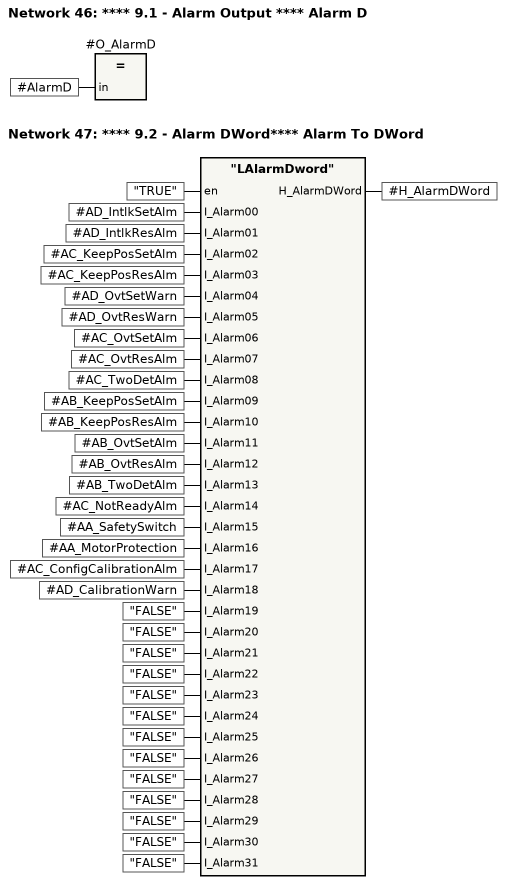
   #O_AlarmD := #AlarmD;
END_REGION

REGION Network 47: **** 9.2 - Alarm DWord**** Alarm To DWord
   // Alarm To DWord
   IF "TRUE" THEN
       "LAlarmDword"(I_Alarm00 := #AD_IntlkSetAlm,
                     I_Alarm01 := #AD_IntlkResAlm,
                     I_Alarm02 := #AC_KeepPosSetAlm,
                     I_Alarm03 := #AC_KeepPosResAlm,
                     I_Alarm04 := #AD_OvtSetWarn,
                     I_Alarm05 := #AD_OvtResWarn,
                     I_Alarm06 := #AC_OvtSetAlm,
                     I_Alarm07 := #AC_OvtResAlm,
                     I_Alarm08 := #AC_TwoDetAlm,
                     I_Alarm09 := #AB_KeepPosSetAlm,
                     I_Alarm10 := #AB_KeepPosResAlm,
                     I_Alarm11 := #AB_OvtSetAlm,
                     I_Alarm12 := #AB_OvtResAlm,
                     I_Alarm13 := #AB_TwoDetAlm,
                     I_Alarm14 := #AC_NotReadyAlm,
                     I_Alarm15 := #AA_SafetySwitch,
                     I_Alarm16 := #AA_MotorProtection,
                     I_Alarm17 := #AC_ConfigCalibrationAlm,
                     I_Alarm18 := #AD_CalibrationWarn,
                     I_Alarm19 := "FALSE",
                     I_Alarm20 := "FALSE",
                     I_Alarm21 := "FALSE",
                     I_Alarm22 := "FALSE",
                     I_Alarm23 := "FALSE",
                     I_Alarm24 := "FALSE",
                     I_Alarm25 := "FALSE",
                     I_Alarm26 := "FALSE",
                     I_Alarm27 := "FALSE",
                     I_Alarm28 := "FALSE",
                     I_Alarm29 := "FALSE",
                     I_Alarm30 := "FALSE",
                     I_Alarm31 := "FALSE",
                     H_AlarmDWord => #H_AlarmDWord);
   END_IF;
END_REGION
END_FUNCTION_BLOCK
